# EPICS substitutions: apps/iocBoot/iocclassc4/joerger_classc4.substitutions
#
# joerger_classc4.substitutions
#
# Author: Wesley Moore (wmoore@jlab.org)
# Date:   Sept 2015
#
file "$(TOP)/db/joerger.db" {
pattern {P,      S,      OUT,        DTYP,               FREQ}
        {frwd_,  scaler, "#C0 S0 @", "Joerger VSC8/16",  10000000}
        {scaler, "",     "#C1 S0 @", "Joerger VSC8/16",  10000000}
}
